// TwinCAT 3 PLC project AxisIaiLibExample
// Title: Test
// Company: Gema
// Author: RG
// ProjectVersion: 0.1.0.0
// ProgramVersion: 3.1.4024.0
// libraries:
//   Tc2_Standard, * (Beckhoff Automation GmbH)
//   Tc2_System, * (Beckhoff Automation GmbH)
//   Tc3_Module, * (Beckhoff Automation GmbH)
//   TcoCore, 0.11.0.35 (Vortex.Library)
//   TcoData, 0.11.0.35 (Vortex.Library)
//   TcoDrivesBeckhoff, 0.11.0.35 (Vortex.Library)
//   TcoElements, 0.11.0.35 (Vortex.Library)
//   TcoInspectors, 0.11.0.29 (Vortex.Library)
//   TcoIo, 0.11.0.35 (Vortex.Library)
//   TcoPneumatics, 0.11.0.35 (Vortex.Library)
//   TcoUtilities, 0.11.0.35 (Vortex.Library)
//   AxisIaiLibrary,0.0.0.1,Gema
// project tree:
//   / PlcTask.TcTTO (not stored)
//   POUs/ AppContext.TcPOU (not stored), MAIN.TcPOU (not stored), MainStation.TcPOU
// real-time tasks:
//   TASK PlcTask: cycle T#10ms, priority 20, ADS port 350

// ---- POUs/MainStation.TcPOU
FUNCTION_BLOCK MainStation EXTENDS TcoCore.TcoObject
VAR
    counter          : INT;

END_VAR

counter := counter + 1;

IF (THIS^.counter MOD 13 = 0) THEN
    THIS^.Messenger.Info('opalalla').Pin();
END_IF

IF (THIS^.counter MOD 400 = 0) THEN
    THIS^.Messenger.Error('ich Poste').Pin();
END_IF

END_FUNCTION_BLOCK
